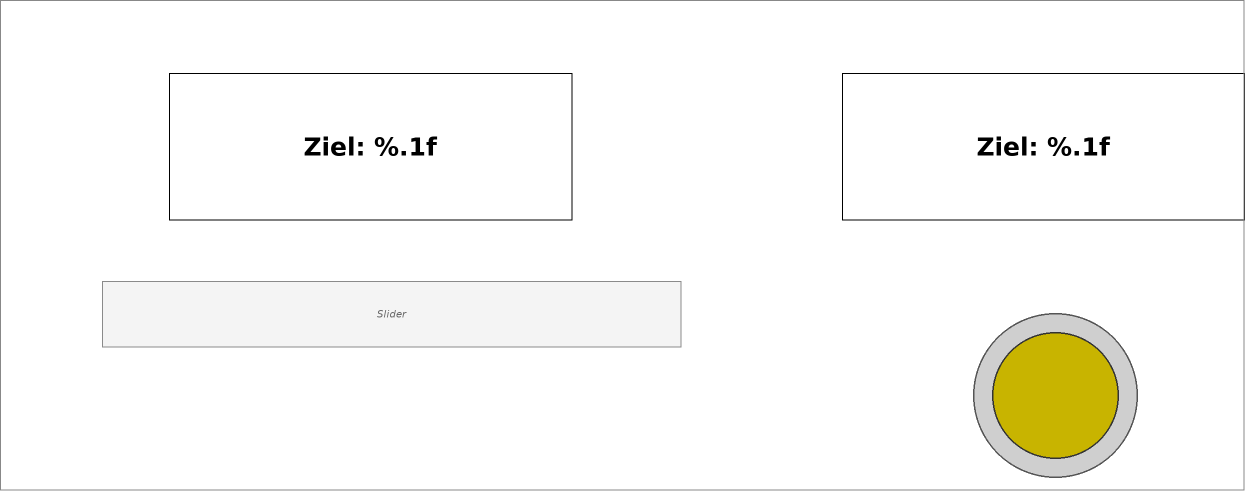
VISUALIZATION Visualization  // 1245x491
    Rectangle (842,73 403x147), "Ziel: %.1f", text variable: MAIN.fTargetValue
        OnMouseClick: write MAIN.fTargetValue via VisuDialogs.Numpad
    Slider (102,281 579x66), variable: MAIN.fActualValue, scale 0..100
    Rectangle (169,73 403x147), "Ziel: %.1f", text variable: MAIN.fActualValue
        OnMouseClick: write MAIN.fTargetValue via VisuDialogs.Numpad
    Lamp1 (956,300 199x191), variable: MAIN.bTargetReached, style: Lamp-Lamp1-Yellow
END_VISUALIZATION

(* stored: Version 1.1.0.1
   Visu Visualization: Id {e5207289-25cd-4cea-a357-4473424b9220} *)
